// TIA Portal V19 export
FUNCTION_BLOCK "Analogue_Input_HMI"   // FB5, LAD
TITLE = Adjust Level Meter From HMI to Control Pump Simulation
{ S7_Optimized_Access := 'TRUE' }
// stored: MemoryReserve 100, SetENOAutomatically false
   VAR_INPUT
      Sensor_Reading { ExternalAccessible := 'False'; ExternalVisible := 'False'; ExternalWritable := 'False'} : Int;   // Reading from Sensor ( on HMI)
   END_VAR
   VAR_OUTPUT
      High_LVL { ExternalAccessible := 'False'; ExternalVisible := 'False'; ExternalWritable := 'False'} : Bool;   // Level High Reached
      Sensor_Reading_Real { ExternalAccessible := 'False'; ExternalVisible := 'False'; ExternalWritable := 'False'} : Real;   // Reading from Sensor (Real)
      Low_LVL { ExternalAccessible := 'False'; ExternalVisible := 'False'; ExternalWritable := 'False'} : Bool;   // Level Low Reached
   END_VAR
   VAR_IN_OUT
      Level_High_SP { ExternalAccessible := 'False'; ExternalVisible := 'False'; ExternalWritable := 'False'} : Real;   // High Level Setpoint Value
      Level_Low_SP { ExternalAccessible := 'False'; ExternalVisible := 'False'; ExternalWritable := 'False'} : Real;   // Low Level Setpoint Value
   END_VAR
BEGIN

REGION Network 1: Convert Int to Real
   // Basic Conversion
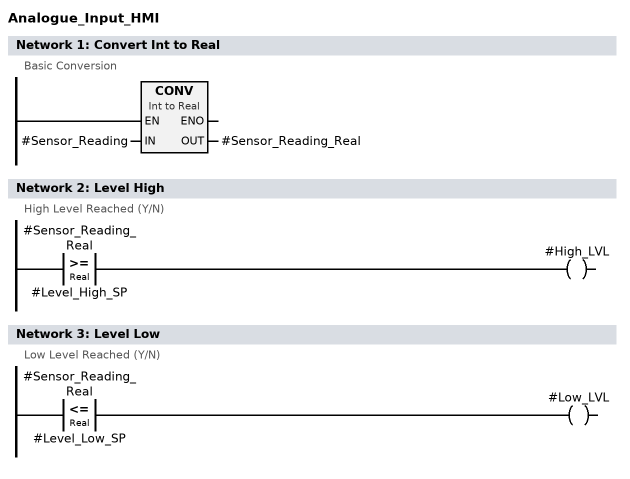
   RUNG wire#powerrail
      { S7_Templates := "[SrcType := Int, DestType := Real]" } Convert(in := #Sensor_Reading, out => #Sensor_Reading_Real)
   END_RUNG
   // the same network as SCL:
   #Sensor_Reading_Real := INT_TO_REAL(#Sensor_Reading);
END_REGION

REGION Network 2: Level High
   // High Level Reached (Y/N)
   RUNG wire#powerrail
      { S7_Templates := "SrcType := Real" } GE_Contact(in1 := #Sensor_Reading_Real, in2 := #Level_High_SP)
      Coil( #High_LVL )
   END_RUNG
   // the same network as SCL:
   #High_LVL := #Sensor_Reading_Real >= #Level_High_SP;
END_REGION

REGION Network 3: Level Low
   // Low Level Reached (Y/N)
   RUNG wire#powerrail
      { S7_Templates := "SrcType := Real" } LE_Contact(in1 := #Sensor_Reading_Real, in2 := #Level_Low_SP)
      Coil( #Low_LVL )
   END_RUNG
   // the same network as SCL:
   #Low_LVL := #Sensor_Reading_Real <= #Level_Low_SP;
END_REGION

REGION Network 4: Spare Network
END_REGION
END_FUNCTION_BLOCK
